(* Logix 5000 project; controller Machine_Maintenance_Lab2 vendor 1 type 14 code 155 rev 36.11; software revision 36.00 *)

TASK MainTask (continuous, watchdog 500 ms) : MainProgram

MODULES
   Local : vendor 1 type 14 code 155 (PointIO 0, rev 36.11)
      Discrete_IO : Embedded (PointIO 1, rev 36.11, Output RPI 20 ms)
END_MODULES

PROGRAM MainProgram   (* main routine MainRoutine *)
VAR
   Count1_High : TIMER := (PRE := 250);
   Count1_Low : TIMER := (PRE := 250);
   Count1_OneShot : BOOL;
   Count1_Pulses : COUNTER := (PRE := 10);
   Count1ON : BOOL;
   Count2_High : TIMER := (PRE := 125);
   Count2_Low : TIMER := (PRE := 125);
   Count2_OneShot : BOOL;
   Count2_Pulses : COUNTER := (PRE := 15);
   Count2ON : BOOL;
   Count3_High : TIMER := (PRE := 500);
   Count3_Low : TIMER := (PRE := 500);
   Count3_OneShot : BOOL;
   Count3_Pulses : COUNTER := (PRE := 6);
   counter : COUNTER := (PRE := 5);
   CycleCounter : COUNTER := (PRE := 5);
   delay : TIMER := (PRE := 10);
   HighCycleTimer : COUNTER := (PRE := 700);
   i_CycleDone : ALIAS FOR o_CycleDone;
   i_GreenPB : ALIAS FOR Local:1:I.Data.0;
   i_GreenPB_ConveyorStart : ALIAS FOR i_GreenPB;
   i_GreenPBLight_Conveyor1ON : ALIAS FOR o_GreenPBLight_Conveyor1ON;
   i_Pause : ALIAS FOR Pause;
   i_Piston : ALIAS FOR Local:1:O.Data.2;
   i_RedPB_StopButton : ALIAS FOR Local:1:I.Data.1;
   i_RedPBLight_Conveyor2ON : ALIAS FOR o_RedPBLight_Conveyor2ON;
   i_Turnkey : ALIAS FOR Local:1:I.Data.2;
   i_Turnkey_ItemSensor : ALIAS FOR i_Turnkey;
   ItemCounter1 : COUNTER := (PRE := 5);
   ItemCounterLeft : COUNTER := (PRE := 5);
   ItemCounterRight : COUNTER := (PRE := 6);
   LowCycleTimer : COUNTER := (PRE := 300);
   NewCycle : BOOL;
   NewCycleCount1 : BOOL;
   NewCycleCount2 : BOOL;
   NewCycleCount3 : BOOL;
   o_CycleDone : BOOL;
   o_GreenPBLight : ALIAS FOR Local:1:O.Data.0;
   o_GreenPBLight_Conveyor1ON : ALIAS FOR o_GreenPBLight;
   o_Piston : ALIAS FOR i_Piston;
   o_RedPBLight : ALIAS FOR Local:1:O.Data.1;
   o_RedPBLight_Conveyor2ON : ALIAS FOR o_RedPBLight;
   OS_Out : BOOL;
   Pause : BOOL;
   Resetcycle3 : BOOL;
   ResetDelay : TIMER := (PRE := 500);
   ResetHigh : BOOL;
   ResetLow : BOOL;
   ThreeSecTimer : TIMER := (PRE := 3000);
   timer : TIMER := (PRE := 5000);
   TimerHighCycle : TIMER := (PRE := 700);
   TimerLowCycle : TIMER := (PRE := 300);
   TurnkeyCounter : COUNTER;
   TurnkeyOneShot : BOOL;
END_VAR
VAR_INPUT
   count1Input : DINT := 10;
   count2input : DINT := 15;
END_VAR

ROUTINE MainRoutine   (* ladder *)
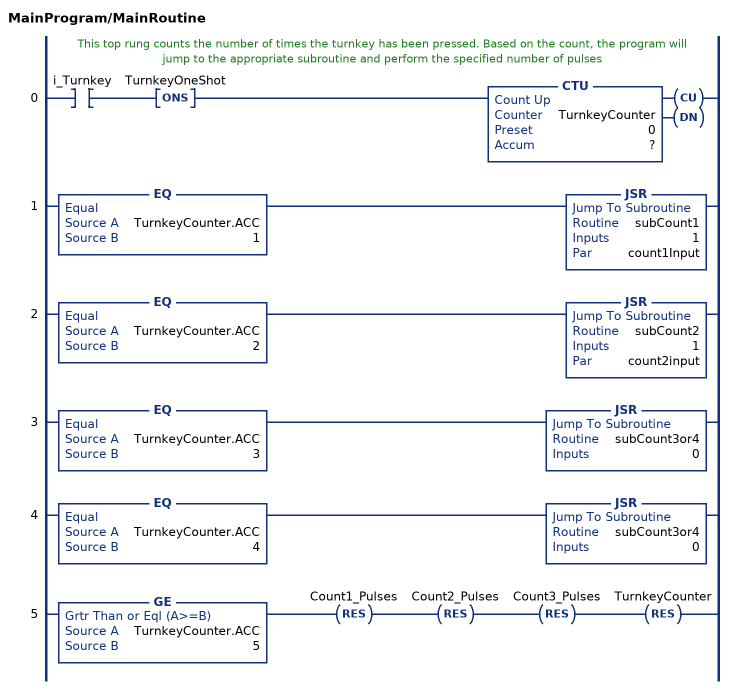
   // This top rung counts the number of times the turnkey has been pressed. Based on the count, the program will jump to the appropriate subroutine and perform the specified number of pulses
   0: XIC(i_Turnkey)ONS(TurnkeyOneShot)CTU(TurnkeyCounter,?,?);
   1: EQ(TurnkeyCounter.ACC,1)JSR(subCount1,1,count1Input);
   2: EQ(TurnkeyCounter.ACC,2)JSR(subCount2,1,count2input);
   3: EQ(TurnkeyCounter.ACC,3)JSR(subCount3or4,0);
   4: EQ(TurnkeyCounter.ACC,4)JSR(subCount3or4,0);
   5: GE(TurnkeyCounter.ACC,5)RES(Count1_Pulses)RES(Count2_Pulses)RES(Count3_Pulses)RES(TurnkeyCounter);
END_ROUTINE

ROUTINE subCount1   (* ladder *)
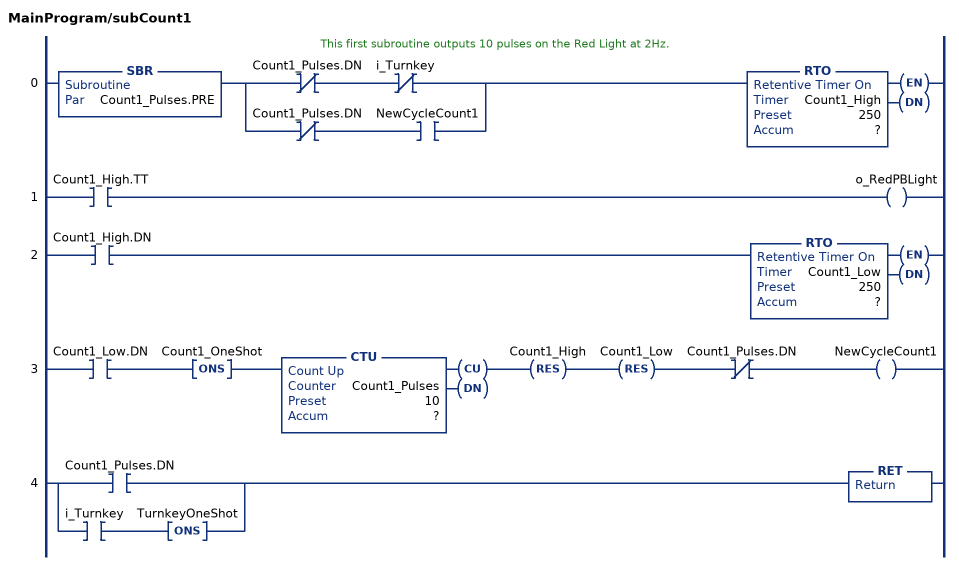
   // This first subroutine outputs 10 pulses on the Red Light at 2Hz.
   0: SBR(Count1_Pulses.PRE)[XIO(Count1_Pulses.DN) XIO(i_Turnkey) ,XIO(Count1_Pulses.DN) XIC(NewCycleCount1) ]RTO(Count1_High,?,?);
   1: XIC(Count1_High.TT)OTE(o_RedPBLight);
   2: XIC(Count1_High.DN)RTO(Count1_Low,?,?);
   3: XIC(Count1_Low.DN)ONS(Count1_OneShot)CTU(Count1_Pulses,?,?)RES(Count1_High)RES(Count1_Low)XIO(Count1_Pulses.DN)OTE(NewCycleCount1);
   4: [XIC(Count1_Pulses.DN) ,XIC(i_Turnkey) ONS(TurnkeyOneShot) ]RET();
END_ROUTINE

ROUTINE subCount2   (* ladder *)
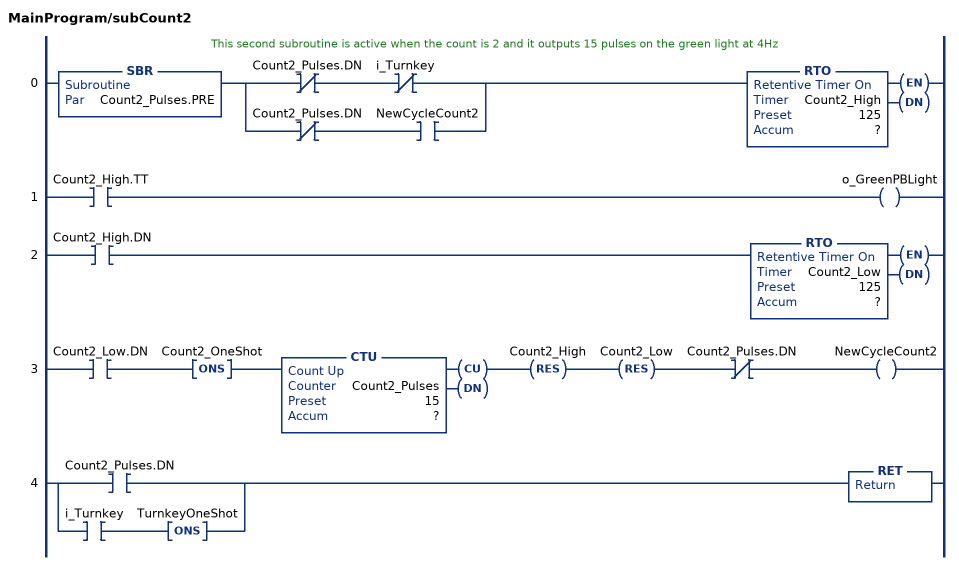
   // This second subroutine is active when the count is 2 and it outputs 15 pulses on the green light at 4Hz
   0: SBR(Count2_Pulses.PRE)[XIO(Count2_Pulses.DN) XIO(i_Turnkey) ,XIO(Count2_Pulses.DN) XIC(NewCycleCount2) ]RTO(Count2_High,?,?);
   1: XIC(Count2_High.TT)OTE(o_GreenPBLight);
   2: XIC(Count2_High.DN)RTO(Count2_Low,?,?);
   3: XIC(Count2_Low.DN)ONS(Count2_OneShot)CTU(Count2_Pulses,?,?)RES(Count2_High)RES(Count2_Low)XIO(Count2_Pulses.DN)OTE(NewCycleCount2);
   4: [XIC(Count2_Pulses.DN) ,XIC(i_Turnkey) ONS(TurnkeyOneShot) ]RET();
END_ROUTINE

ROUTINE subCount3or4   (* ladder *)
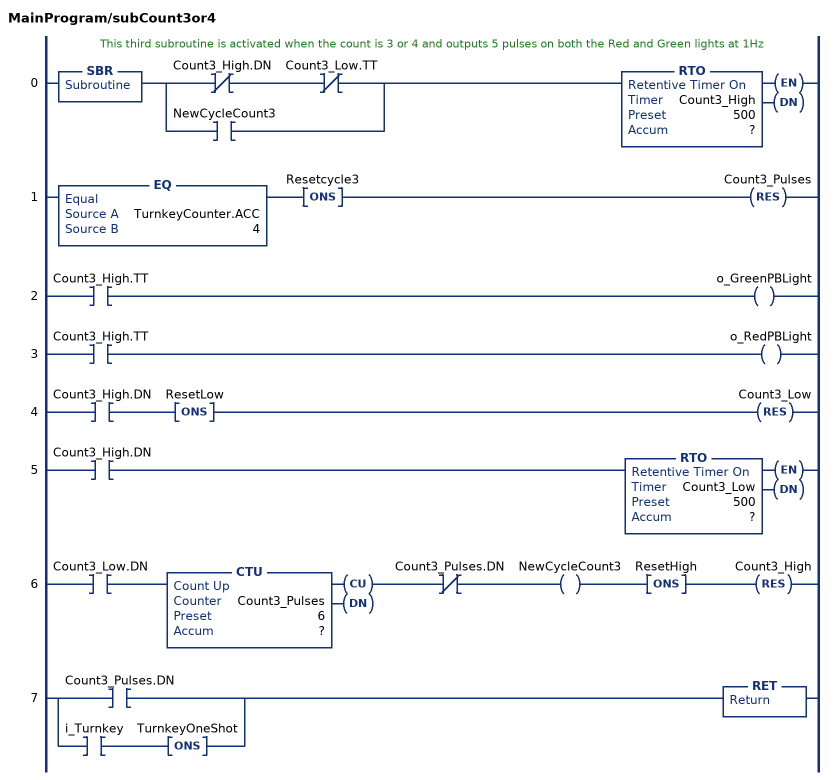
   // This third subroutine is activated when the count is 3 or 4 and outputs 5 pulses on both the Red and Green lights at 1Hz
   0: SBR()[XIO(Count3_High.DN) XIO(Count3_Low.TT) ,XIC(NewCycleCount3) ]RTO(Count3_High,?,?);
   1: EQ(TurnkeyCounter.ACC,4)ONS(Resetcycle3)RES(Count3_Pulses);
   2: XIC(Count3_High.TT)OTE(o_GreenPBLight);
   3: XIC(Count3_High.TT)OTE(o_RedPBLight);
   4: XIC(Count3_High.DN)ONS(ResetLow)RES(Count3_Low);
   5: XIC(Count3_High.DN)RTO(Count3_Low,?,?);
   6: XIC(Count3_Low.DN)CTU(Count3_Pulses,?,?)XIO(Count3_Pulses.DN)OTE(NewCycleCount3)ONS(ResetHigh)RES(Count3_High);
   7: [XIC(Count3_Pulses.DN) ,XIC(i_Turnkey) ONS(TurnkeyOneShot) ]RET();
END_ROUTINE
END_PROGRAM
